{attribute 'qualified_only'}
VAR_GLOBAL CONSTANT
	MAX_SIZE_MSG_TO_SEND	:UINT := 1000;
	MAX_SIZE_MSG_TO_RCV		:UINT := 1000;
END_VAR

(* stored: Version 1.1.0.1
   GVL P_AmeClt: Id {577cfc17-fe10-057e-0c17-021c822b11b9}, ParameterList True *)
